FUNCTION_BLOCK SafetyMotionBlockingWidget
VAR_INPUT
END_VAR
VAR_OUTPUT
	actualStatus : StatusWidget;
END_VAR
VAR_IN_OUT
	ref : SafetyMotionBlocking;
END_VAR
VAR
END_VAR


actualStatus(text  := ref.actualStatus,
             color := HealthToColor(ref.statuses.healthStatus));

END_FUNCTION_BLOCK

(* stored: Version 1.1.0.1, ProductVersion 3.1.4018.5
   POU SafetyMotionBlockingWidget: Id {4f135694-d524-4cc0-9ade-3f014d523e55}, SpecialFunc None *)
